FUNCTION_BLOCK FB_NOTT_CALIBRATION_BEAM_SPLITTER
VAR_INPUT
END_VAR
VAR_OUTPUT
END_VAR
VAR
	NBS:		FB_NOTT_MOTOR;
	
	SIM_NBS:	FB_SIM_MOTOR;
	
	stat:		T_NOTT_STAT;
END_VAR



NBS(
	in_bSafe:=, 
	in_bDisableIfUnsafe:=, 
	sName:= 'NBS', 
	nNOVRAM_DevId:= 6, 
	nNOVRAM_Offset:= 37000);
	
SIM_NBS (ptrCfg:=ADR(NBS.cfg), ptrStat:=ADR(NBS.stat));

END_FUNCTION_BLOCK

(* stored: Version 1.1.0.1, ProductVersion 3.1.4024.14
   POU FB_NOTT_CALIBRATION_BEAM_SPLITTER: Id {ffb51bfc-3265-4bf1-a72e-e51bc2ac613c}, SpecialFunc None *)
